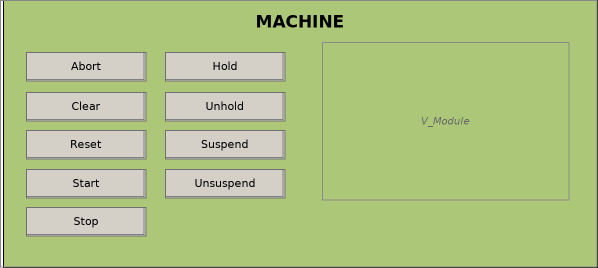
VISUALIZATION V_MachineModule  // 598x268
VAR_IN_OUT
	HMI : ST_PackMLBaseModule_HMI;
END_VAR
    Group (3,0 595x268)
        RoundedRectangle (0,0 595x268)
        Button (23,52 120x29), "Abort"
            OnMouseClick: execute { HMI.Command.State := E_PMLCommand.ePMLCommand_Abort; }
        Button (23,92 120x29), "Clear"
            OnMouseClick: execute { HMI.Command.State := E_PMLCommand.ePMLCommand_Clear; }
        Button (23,130 120x29), "Reset"
            OnMouseClick: execute { HMI.Command.State := E_PMLCommand.ePMLCommand_Reset; }
        Button (23,169 120x29), "Start"
            OnMouseClick: execute { HMI.Command.State := E_PMLCommand.ePMLCommand_Start; }
        Button (23,207 120x29), "Stop"
            OnMouseClick: execute { HMI.Command.State := E_PMLCommand.ePMLCommand_Stop; }
        Button (162,52 120x29), "Hold"
            OnMouseClick: execute { HMI.Command.State := E_PMLCommand.ePMLCommand_Hold; }
        Button (162,92 120x29), "Unhold"
            OnMouseClick: execute { HMI.Command.State := E_PMLCommand.ePMLCommand_Unhold; }
        Button (162,130 120x29), "Suspend"
            OnMouseClick: execute { HMI.Command.State := E_PMLCommand.ePMLCommand_Suspend; }
        Button (162,169 120x29), "Unsuspend"
            OnMouseClick: execute { HMI.Command.State := E_PMLCommand.ePMLCommand_Unsuspend; }
        Frame (319,42 247x158)
            shows V_Module(HMI := HMI)
    Label (15,3 570x37), "MACHINE"
END_VISUALIZATION

(* stored: Version 1.1.0.1, ProductVersion 3.1.4024.16
   Visu V_MachineModule: Id {38d3adcf-05a5-497d-bb81-55443dba2d43} *)
